{attribute 'Tc2GvlVarNames'}
{attribute 'strict'}
//Tipologia Funzionamento Macchina
TYPE e_Tipo_Funzionamento :
(
	NOT_DEFINED							:= -1, 	(* Tipologia Indefinita *)
	FUNZIONAMENTO_PALLETTIZZATORE	 	:= 0,	(* Tipologia di Funzionamento di Tipo Pallettizzatore: Prelievo Da Linea Classico *)
	FUNZIONAMENTO_PICKING				:= 1,	(* Tipologia di Funzionamento di Tipo Pallettizzatore: Prelievo e Deposito in Postazione *)
	FUNZIONAMENTO_MISTO					:= 2, 	(* Tipologia di Funzionamento di Tipo Pallettizzatore: Prelievo Da Linea Classico + Prelievo e Deposito in Postazione *)
	FUNZIONAMENTO_DEPAL					:= 3, 	(* Tipologia di Funzionamento di Tipo Depallettizzatore: Prelevo da una postazione con cavallina, cassa o pallet e appoggio sulla linea *)
	FUNZIONAMENTO_SLAVE					:= 4	(* Tipologia di Funzionamento di Tipo SLAVE: la macchina esegue le missioni che gli vengono dettate da un ente esterno (WMS)*)

);
END_TYPE
//  NOT_DEFINED = '-1'

(* stored: Version 1.1.0.1, ProductVersion 3.1.4024.11
   EnumerationTextList e_Tipo_Funzionamento: Id {dd3e8eb6-a3fe-4587-8a83-3f44a9fbe315} *)
